(*
  QualiVision line camera system
  DMAX106.   
*)
FUNCTION_BLOCK FB_LineCamera106 EXTENDS FB_LineCamera

VAR CONSTANT
  cCameraWidth106           : DINT := 13440;   (*Camera width [px]*)
  cCameraMechOffsetTC106    : REAL :=  88.0;   (*Camera mechanical offset at calibration temp [mm]*)
  cMechOffsetCameraToPU106  : REAL :=  30.31;  (*Camera mechanical offset to PrintUnit [mm]*)
  cPrintUnitMechOffsetTC106 : REAL := 31.4747; (*PrintUnit mechanical offset at calibration temp [mm]*)
END_VAR

SUPER^();

METHOD InitLineCamera
VAR_INPUT
  nPrintUnitResolution         : UDINT;    (*printhead pixel resolution [dpi]*)
  nPrintUnitSubPx              : UDINT;    (*print unit subPixel resolution [SubPx]*)
  nPrintUnitWidth              : UDINT;    (*print unit width in [px]*)
  iCameraTrigger               : I_CameraTrigger;
END_VAR
(*Init for dmax type*)
_nCameraWidth           := cCameraWidth106;
_fCameraMechOffsetTC    := cCameraMechOffsetTC106;
_fMechOffsetCameraToPU  := cMechOffsetCameraToPU106;
_fPrintUnitMechOffsetTC := cPrintUnitMechOffsetTC106;

SUPER^.InitLineCamera( nPrintUnitResolution := nPrintUnitResolution
                      , nPrintUnitSubPx := nPrintUnitSubPx
                      , nPrintUnitWidth := nPrintUnitWidth
                      , iCameraTrigger := iCameraTrigger);
END_METHOD

{attribute 'monitoring':='variable'}
PROPERTY sName : STRING
GET
sName := 'LineCam 106';
END_GET
END_PROPERTY

END_FUNCTION_BLOCK

(* stored: Version 1.1.0.1, ProductVersion 3.1.4024.3
   POU FB_LineCamera106: Id {e2ca7b23-5d9c-4a28-90a4-190f0095c257}, SpecialFunc None
   Method InitLineCamera: Id {6d78d247-28ed-444e-9902-ffe57fa67cbc}
   Property sName: Id {d882d9f0-4b80-45f3-b121-98e01ebf8c13}
   Get Get: Id {aae23f89-016d-49be-b465-f87827d4de86} *)
